TYPE U_NCI_R_PARAMETER_I :
UNION

  stCtrl              : ARRAY[1..MAX_NCI_CH] OF ST_R_Parameter;

  byCtrl    AT %I*    : ARRAY[1..MAX_NCI_CH] OF
                        ARRAY[1..SIZEOF(ST_R_Parameter)] OF BYTE;
END_UNION
END_TYPE

(* stored: Version 1.1.0.1, ProductVersion 3.1.4026.13
   DUT U_NCI_R_PARAMETER_I: Id {9a3d6383-9d4b-472a-a2eb-49c6062ddf1b} *)
